// TIA Portal V19 export
TYPE "LEXCHANGETRAY_typeScanner_hmiInterface"
// stored: Access Published
   STRUCT
      monitor : "LEXCHANGETRAY_typeScanner_monitor";
      sim { S7_SetPoint := 'True'} : "LEXCHANGETRAY_typeScanner_sim";
   END_STRUCT;
END_TYPE
